{attribute wpf [Container(Layout.Scroll)]}
TYPE Scroll_other :
STRUCT
	{attribute wpf [Container(Layout.Stack)]}
	_wheel_stack: Wheel;
	{attribute wpf [Container(Layout.UniformGrid)]}
	_wheel_ug: Wheel;
	{attribute wpf [Container(Layout.Wrap)]}
	_wheel_wrap: Wheel;
	{attribute wpf [Container(Layout.Tabs)]}
	_wheel_tabs: Wheel;
	{attribute wpf [Container(Layout.Border)]}
	_wheel_border: Wheel;
	{attribute wpf [Container(Layout.GroupBox)]}
	_wheel_gb: Wheel;
END_STRUCT
END_TYPE

(* stored: Version 1.1.0.1, ProductVersion 3.1.4024.9
   DUT Scroll_other: Id {183fd1c7-3942-4dbe-97a7-bb2908a8a151} *)
